(* Logix 5000 project; controller ABB_Drive_Test vendor 1 type 14 code 149 rev 33.12; software revision 33.01; part 3 of 6 *)
(* tags used below, declared in another part *)
   CF0x3MSG : MESSAGE;   // detect card
   CF0x4fMSG : MESSAGE;   // read from file
   CF0x50MSG : MESSAGE;   // write to file
   CF0x52MSG : MESSAGE;   // file open
   CF0x53MSG : MESSAGE;   // set file pointer
   CF0x54MSG : MESSAGE;   // file close
   CF0x55MSG : MESSAGE;   // delete file
   CF0x56MSG : MESSAGE;   // create directory
   CF0x57MSG : MESSAGE;   // rename/move file
   CF0x58MSG : MESSAGE;   // Find first file
   CF0x59MSG : MESSAGE;   // Find next file
   CF0x5aMSG : MESSAGE;   // Find close
   CF_data : SINT[512];
   CF_RW_functions : CF_functions;

PROGRAM CF_FunctionsProgram   (* main routine MainRoutine *)
// version 3
// june 2014
VAR
   append : BOOL := 1;
   bytestring : STRING := ' KB';
   CF_del : TIMER := (PRE := 5);
   cmd_timeout : TIMER := (PRE := 4000);
   cmdto : BOOL;
   dir_only : BOOL;
   extra_info : BOOL;
   f_nr : DINT := 75;
   falctrl01 : CONTROL := (LEN := 81, POS := 80, EN := 1, DN := 1);
   filehandle : DINT;
   flush_delay : TIMER := (PRE := 500);
   intsource : INT[100] := ([0] := 24, [1] := 76, [2] := 111, [3] := 103, [4] := 95, [5] := 49, [6] := 57, [7] := 57, [8] := 56, [9] := 95, [10] := 48, [11] := 52, [12] := 95, [13] := 48, [14] := 51, [15] := 95, [16] := 48, [17] := 50, [18] := 95, [19] := 49, [20] := 49, [21] := 46, [22] := 99, [23] := 115, [24] := 118);
   MSGtriggers : DINT;
        .0   // 0x4f
        .1   // 0x50
        .10   // 0x59
        .11   // 0x5a
        .2   // 0x51
        .3   // 0x52
        .4   // 0x53
        .5   // 0x54
        .6   // 0x55
        .7   // 0x56
        .8   // 0x57
        .9   // 0x58
   next_file_response : FS_response := (pot_holder := -242345696, fflags := 16#0000_0020, create_TS := 125357957340000000, last_write_TS := 125357957340000000, size := 252800, name[0] := '$00$18', name[1] := '$00L', name[2] := '$00o', name[3] := '$00g', name[4] := '$00_', name[5] := '$001', name[6] := '$009', name[7] := '$009', name[8] := '$008', name[9] := '$00_', name[10] := '$000', name[11] := '$003', name[12] := '$00_', name[13] := '$003', name[14] := '$001', name[15] := '$00_', name[16] := '$000', name[17] := '$004', name[18] := '$00_', name[19] := '$005', name[20] := '$005', name[21] := '$00.', name[22] := '$00c', name[23] := '$00s', name[24] := '$00v', name[25] := '$00s', name[26] := '$00v', name[27] := '8,', name[28] := '0.', name[29] := '00', name[30] := '00', name[31] := '00', name[32] := ',0', name[33] := '.9', name[34] := '00', name[35] := '00', name[36] := '00', name[37] := '00', name[38] := '1,', name[39] := '.0', name[40] := '00', name[41] := '00', name[42] := '00', name[43] := ',0', name[44] := '11', name[45] := '0.', name[46] := '00', name[47] := '00', name[48] := '00', name[49] := '1,', name[50] := '.2', name[51] := '00', name[52] := '00', name[53] := '00', name[54] := ',0',
        name[55] := '.1', name[56] := '00', name[57] := '00', name[58] := '00', name[59] := '00', name[60] := '$0A$0D', name[61] := '53', name[62] := '88', name[63] := ',8', name[64] := '.0', name[65] := '90', name[66] := '31', name[67] := '71', name[68] := '07', name[69] := '2,', name[70] := '0.', name[71] := '00', name[72] := '00', name[73] := '00', name[74] := ',0', name[75] := '.5', name[76] := '00', name[77] := '00', name[78] := '00', name[79] := '00', name[80] := '6,', name[81] := '0.', name[82] := '00', name[83] := '00', name[84] := '00', name[85] := ',0', name[86] := '.7', name[87] := '00', name[88] := '00', name[89] := '00', name[90] := '00', name[91] := '8,', name[92] := '0.', name[93] := '00', name[94] := '00', name[95] := '00', name[96] := ',0', name[97] := '.9', name[98] := '00', name[99] := '00');
        .fflags.0   // Read Only
        .fflags.1   // Hidden
        .fflags.2   // System
   prev_index : DINT := 10;
   searchstring : STRING := 'Log_1998_04_03_02_11.csv';
   slot_number : DINT;
   spacestring : STRING := '        ';
   step : DINT;
   step_copy : DINT := 99;
   tempDINT : DINT := 392;
   tempDINTAR : DINT[10] := ([0] := 1073741824, [3] := 4, [4] := 128, [7] := 40, [8] := 20224);
   tempstring : STRING := '$01$00';
END_VAR

ROUTINE ascii2uni   (* ladder *)
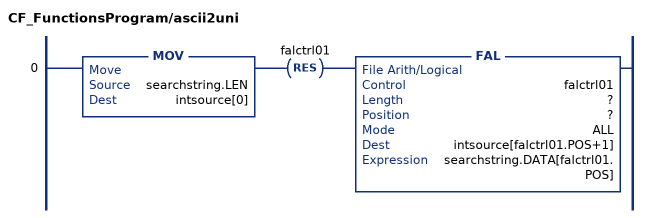
   0: MOV(searchstring.LEN,intsource[0])RES(falctrl01)FAL(falctrl01,?,?,ALL,intsource[falctrl01.POS+1],searchstring.DATA[falctrl01.POS]);
END_ROUTINE

ROUTINE MainRoutine   (* ladder *)
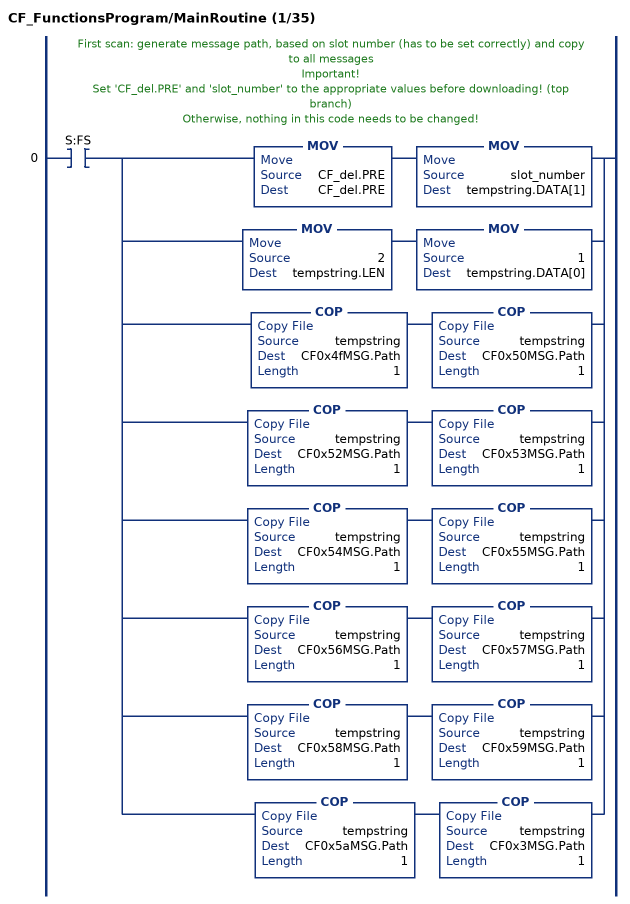
   // First scan: generate message path, based on slot number (has to be set correctly) and copy to all messages
   // Important!
   // Set 'CF_del.PRE' and 'slot_number' to the appropriate values before downloading! (top branch)
   // Otherwise, nothing in this code needs to be changed!
   0: XIC(S:FS)[MOV(CF_del.PRE,CF_del.PRE) MOV(slot_number,tempstring.DATA[1]) ,MOV(2,tempstring.LEN) MOV(1,tempstring.DATA[0]) ,COP(tempstring,CF0x4fMSG.Path,1) COP(tempstring,CF0x50MSG.Path,1) ,COP(tempstring,CF0x52MSG.Path,1) COP(tempstring,CF0x53MSG.Path,1) ,COP(tempstring,CF0x54MSG.Path,1) COP(tempstring,CF0x55MSG.Path,1) ,COP(tempstring,CF0x56MSG.Path,1) COP(tempstring,CF0x57MSG.Path,1) ,COP(tempstring,CF0x58MSG.Path,1) COP(tempstring,CF0x59MSG.Path,1) ,COP(tempstring,CF0x5aMSG.Path,1) COP(tempstring,CF0x3MSG.Path,1) ];
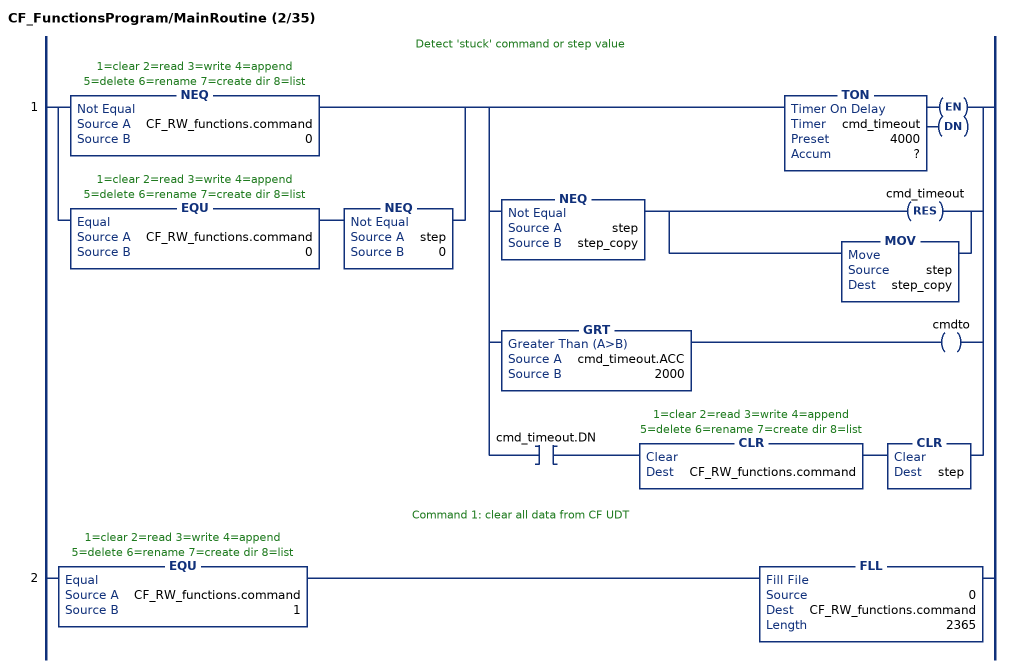
   // Detect 'stuck' command or step value
   1: [NEQ(CF_RW_functions.command,0) ,EQU(CF_RW_functions.command,0) NEQ(step,0) ][TON(cmd_timeout,?,?) ,NEQ(step,step_copy) [RES(cmd_timeout) ,MOV(step,step_copy) ] ,GRT(cmd_timeout.ACC,2000) OTE(cmdto) ,XIC(cmd_timeout.DN) CLR(CF_RW_functions.command) CLR(step) ];
   // Command 1: clear all data from CF UDT
   2: EQU(CF_RW_functions.command,1)FLL(0,CF_RW_functions.command,2365);
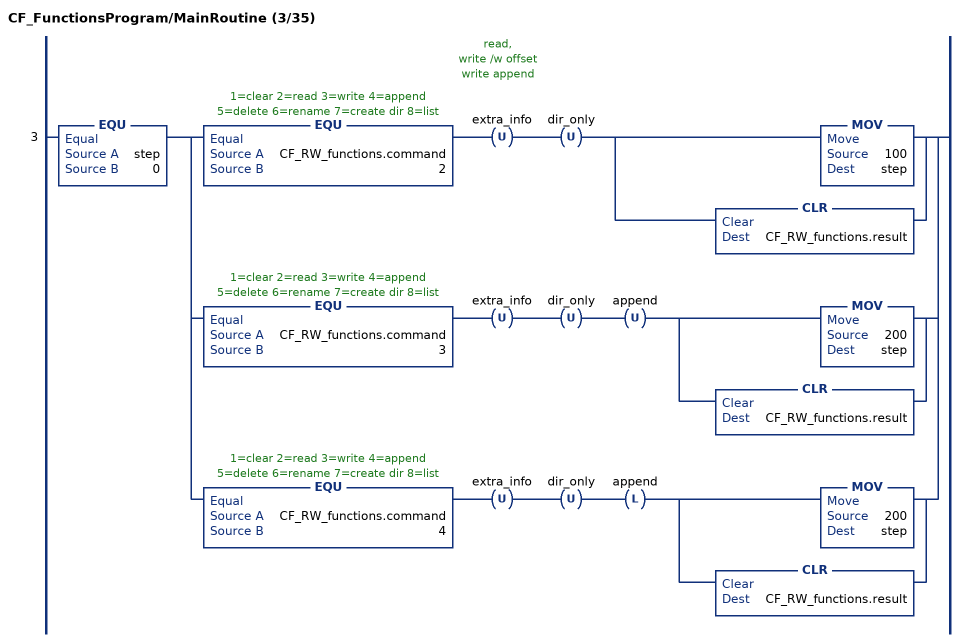
   // read,
   // write /w offset
   // write append
   3: EQU(step,0)[EQU(CF_RW_functions.command,2) OTU(extra_info) OTU(dir_only) [MOV(100,step) ,CLR(CF_RW_functions.result) ] ,EQU(CF_RW_functions.command,3) OTU(extra_info) OTU(dir_only) OTU(append) [MOV(200,step) ,CLR(CF_RW_functions.result) ] ,EQU(CF_RW_functions.command,4) OTU(extra_info) OTU(dir_only) OTL(append) [MOV(200,step) ,CLR(CF_RW_functions.result) ] ];
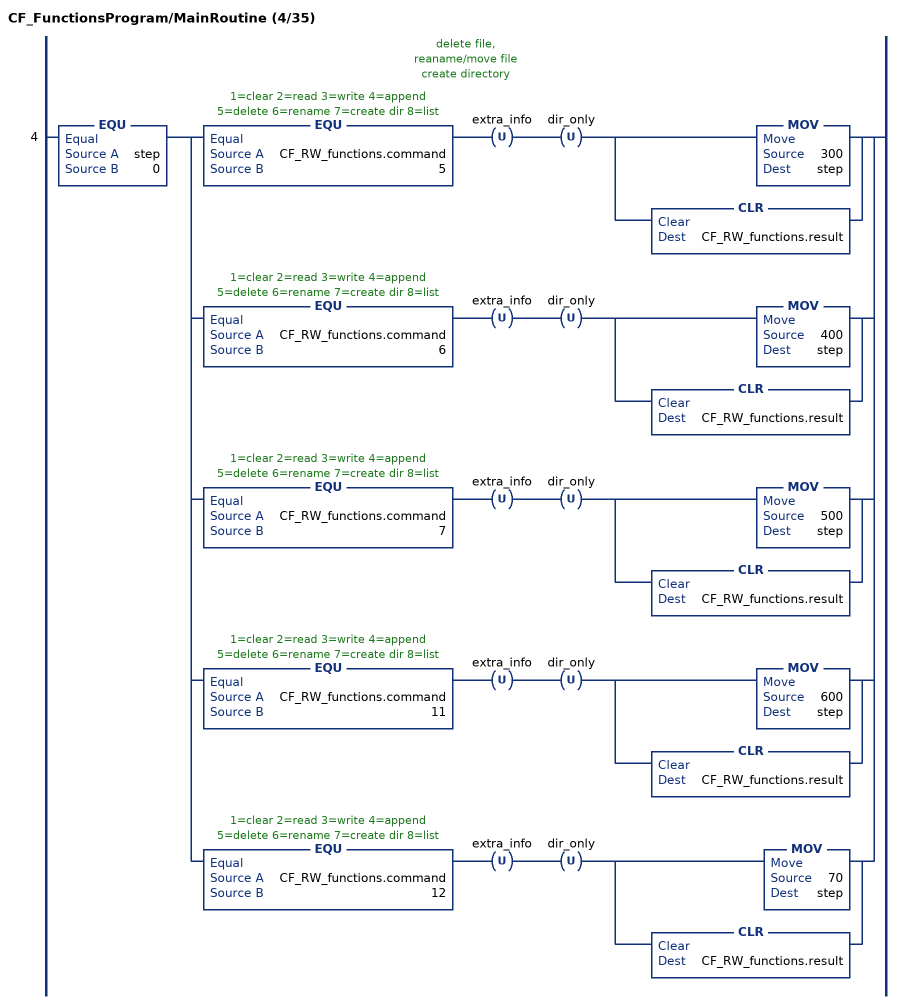
   // delete file,
   // reaname/move file
   // create directory
   4: EQU(step,0)[EQU(CF_RW_functions.command,5) OTU(extra_info) OTU(dir_only) [MOV(300,step) ,CLR(CF_RW_functions.result) ] ,EQU(CF_RW_functions.command,6) OTU(extra_info) OTU(dir_only) [MOV(400,step) ,CLR(CF_RW_functions.result) ] ,EQU(CF_RW_functions.command,7) OTU(extra_info) OTU(dir_only) [MOV(500,step) ,CLR(CF_RW_functions.result) ] ,EQU(CF_RW_functions.command,11) OTU(extra_info) OTU(dir_only) [MOV(600,step) ,CLR(CF_RW_functions.result) ] ,EQU(CF_RW_functions.command,12) OTU(extra_info) OTU(dir_only) [MOV(70,step) ,CLR(CF_RW_functions.result) ] ];
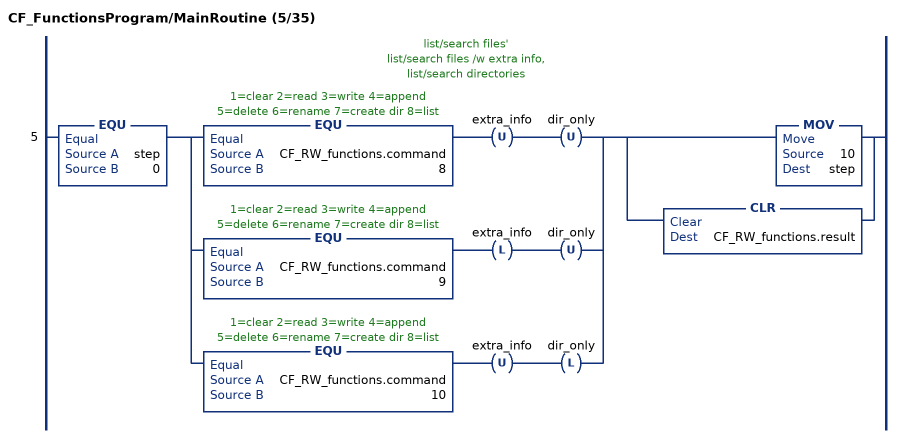
   // list/search files'
   // list/search files /w extra info,
   // list/search directories
   5: EQU(step,0)[EQU(CF_RW_functions.command,8) OTU(extra_info) OTU(dir_only) ,EQU(CF_RW_functions.command,9) OTL(extra_info) OTU(dir_only) ,EQU(CF_RW_functions.command,10) OTU(extra_info) OTL(dir_only) ][MOV(10,step) ,CLR(CF_RW_functions.result) ];
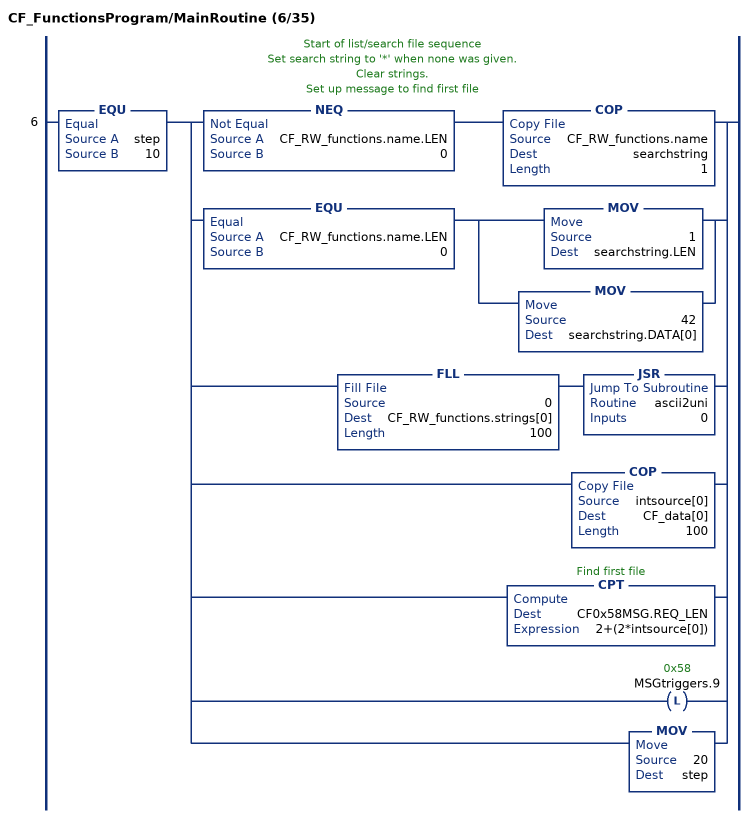
   // Start of list/search file sequence
   //  Set search string to '*' when none was given.
   // Clear strings.
   // Set up message to find first file
   6: EQU(step,10)[NEQ(CF_RW_functions.name.LEN,0) COP(CF_RW_functions.name,searchstring,1) ,EQU(CF_RW_functions.name.LEN,0) [MOV(1,searchstring.LEN) ,MOV(42,searchstring.DATA[0]) ] ,FLL(0,CF_RW_functions.strings[0],100) JSR(ascii2uni,0) ,COP(intsource[0],CF_data[0],100) ,CPT(CF0x58MSG.REQ_LEN,2+(2*intsource[0])) ,OTL(MSGtriggers.9) ,MOV(20,step) ];
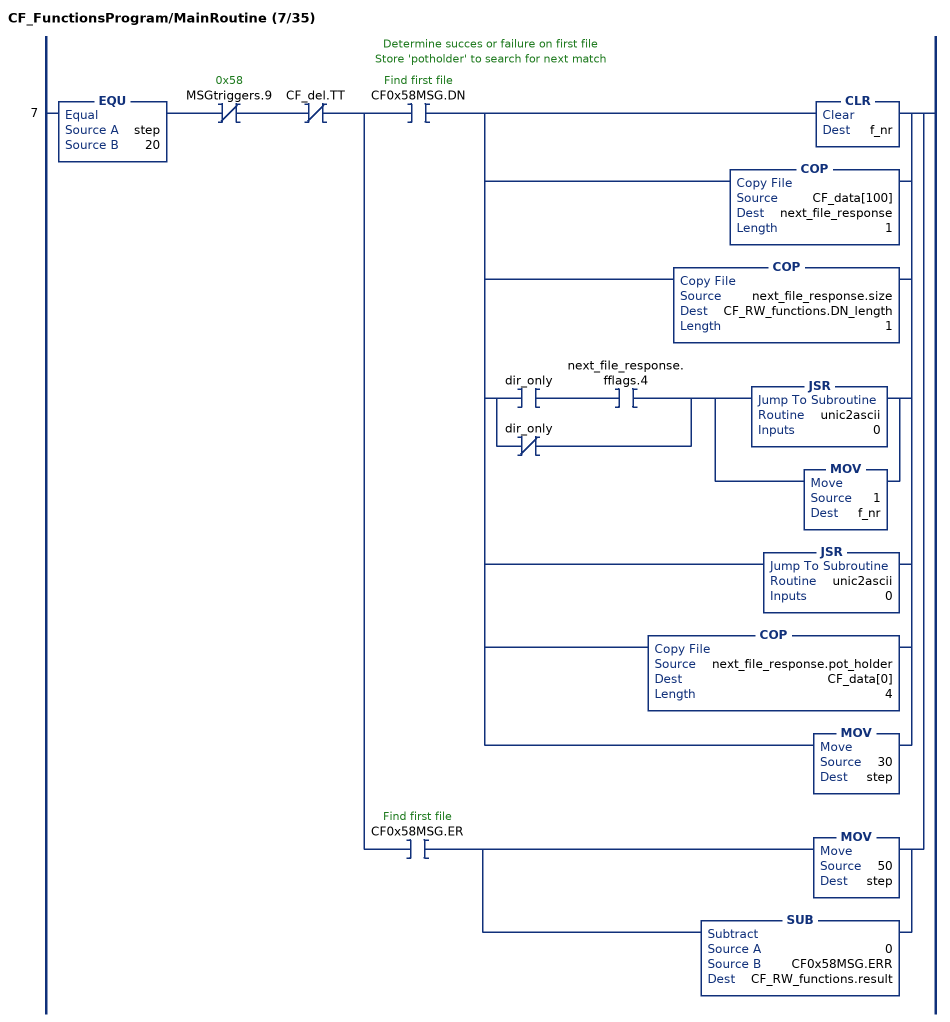
   // Determine succes or failure on first file
   // Store 'potholder' to search for next match
   7: EQU(step,20)XIO(MSGtriggers.9)XIO(CF_del.TT)[XIC(CF0x58MSG.DN) [CLR(f_nr) ,COP(CF_data[100],next_file_response,1) ,COP(next_file_response.size,CF_RW_functions.DN_length,1) ,[XIC(dir_only) XIC(next_file_response.fflags.4) ,XIO(dir_only) ] [JSR(unic2ascii,0) ,MOV(1,f_nr) ] ,JSR(unic2ascii,0) ,COP(next_file_response.pot_holder,CF_data[0],4) ,MOV(30,step) ] ,XIC(CF0x58MSG.ER) [MOV(50,step) ,SUB(0,CF0x58MSG.ERR,CF_RW_functions.result) ] ];
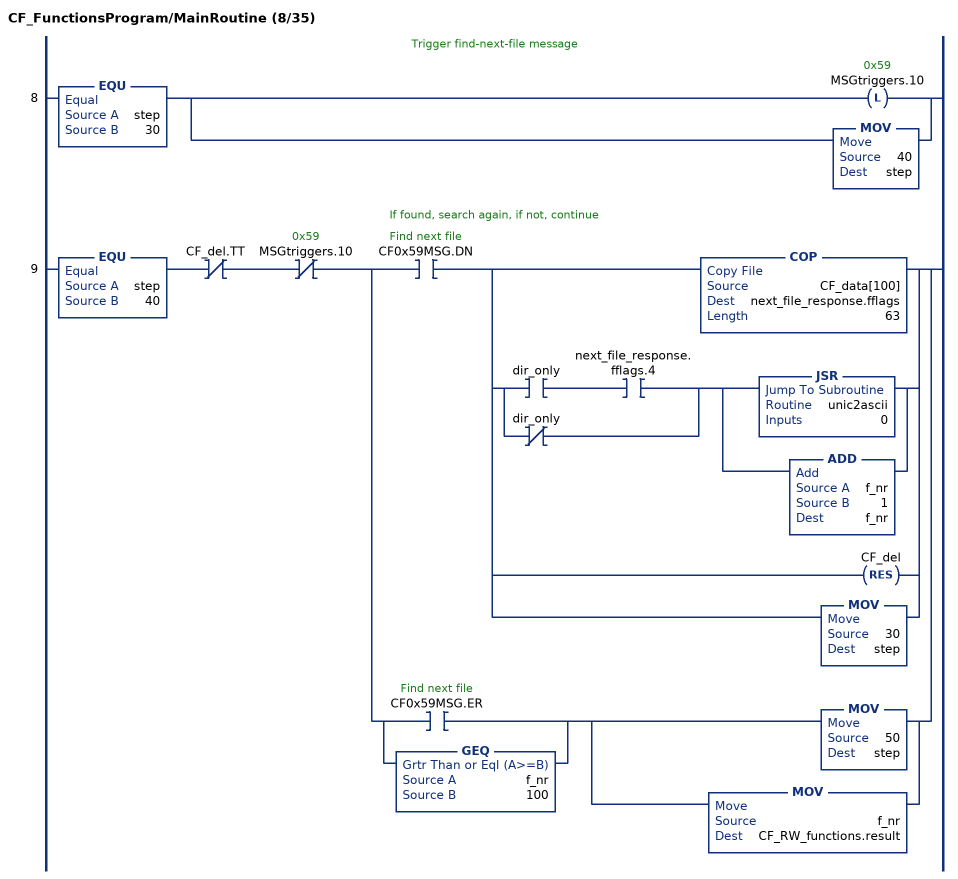
   // Trigger find-next-file message
   8: EQU(step,30)[OTL(MSGtriggers.10) ,MOV(40,step) ];
   // If found, search again, if not, continue
   9: EQU(step,40)XIO(CF_del.TT)XIO(MSGtriggers.10)[XIC(CF0x59MSG.DN) [COP(CF_data[100],next_file_response.fflags,63) ,[XIC(dir_only) XIC(next_file_response.fflags.4) ,XIO(dir_only) ] [JSR(unic2ascii,0) ,ADD(f_nr,1,f_nr) ] ,RES(CF_del) ,MOV(30,step) ] ,[XIC(CF0x59MSG.ER) ,GEQ(f_nr,100) ] [MOV(50,step) ,MOV(f_nr,CF_RW_functions.result) ] ];
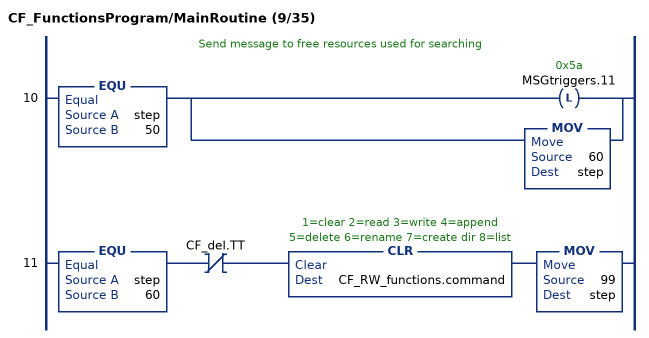
   // Send message to free resources used for searching
   10: EQU(step,50)[OTL(MSGtriggers.11) ,MOV(60,step) ];
   11: EQU(step,60)XIO(CF_del.TT)CLR(CF_RW_functions.command)MOV(99,step);
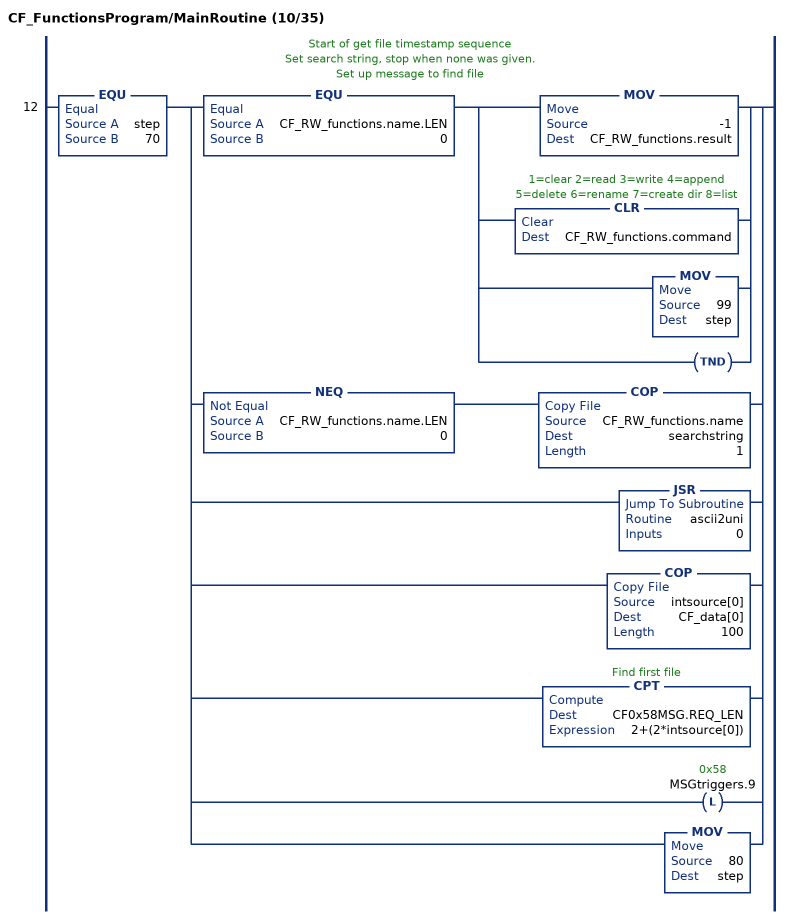
   // Start of get file timestamp sequence
   //  Set search string, stop when none was given.
   // Set up message to find file
   12: EQU(step,70)[EQU(CF_RW_functions.name.LEN,0) [MOV(-1,CF_RW_functions.result) ,CLR(CF_RW_functions.command) ,MOV(99,step) ,TND() ] ,NEQ(CF_RW_functions.name.LEN,0) COP(CF_RW_functions.name,searchstring,1) ,JSR(ascii2uni,0) ,COP(intsource[0],CF_data[0],100) ,CPT(CF0x58MSG.REQ_LEN,2+(2*intsource[0])) ,OTL(MSGtriggers.9) ,MOV(80,step) ];
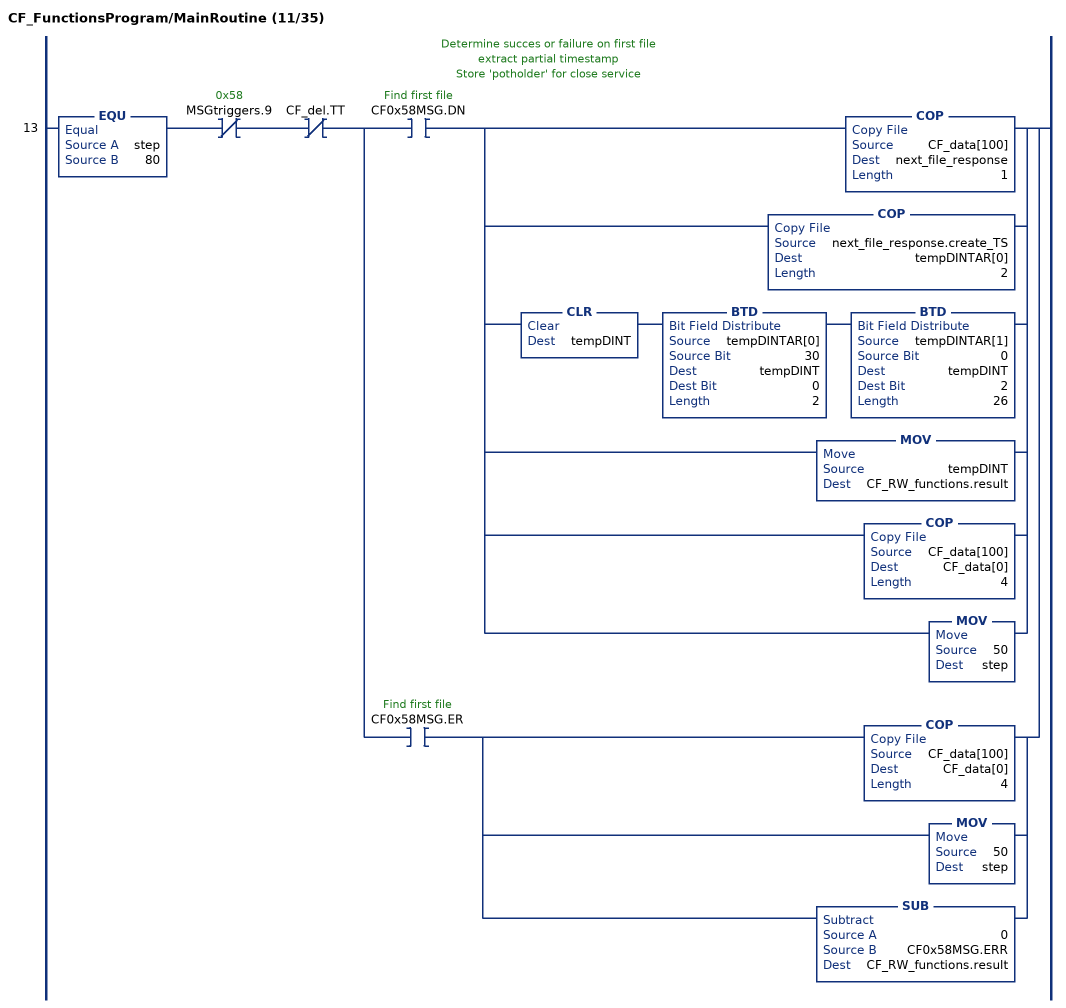
   // Determine succes or failure on first file
   // extract partial timestamp
   // Store 'potholder' for close service
   13: EQU(step,80)XIO(MSGtriggers.9)XIO(CF_del.TT)[XIC(CF0x58MSG.DN) [COP(CF_data[100],next_file_response,1) ,COP(next_file_response.create_TS,tempDINTAR[0],2) ,CLR(tempDINT) BTD(tempDINTAR[0],30,tempDINT,0,2) BTD(tempDINTAR[1],0,tempDINT,2,26) ,MOV(tempDINT,CF_RW_functions.result) ,COP(CF_data[100],CF_data[0],4) ,MOV(50,step) ] ,XIC(CF0x58MSG.ER) [COP(CF_data[100],CF_data[0],4) ,MOV(50,step) ,SUB(0,CF0x58MSG.ERR,CF_RW_functions.result) ] ];
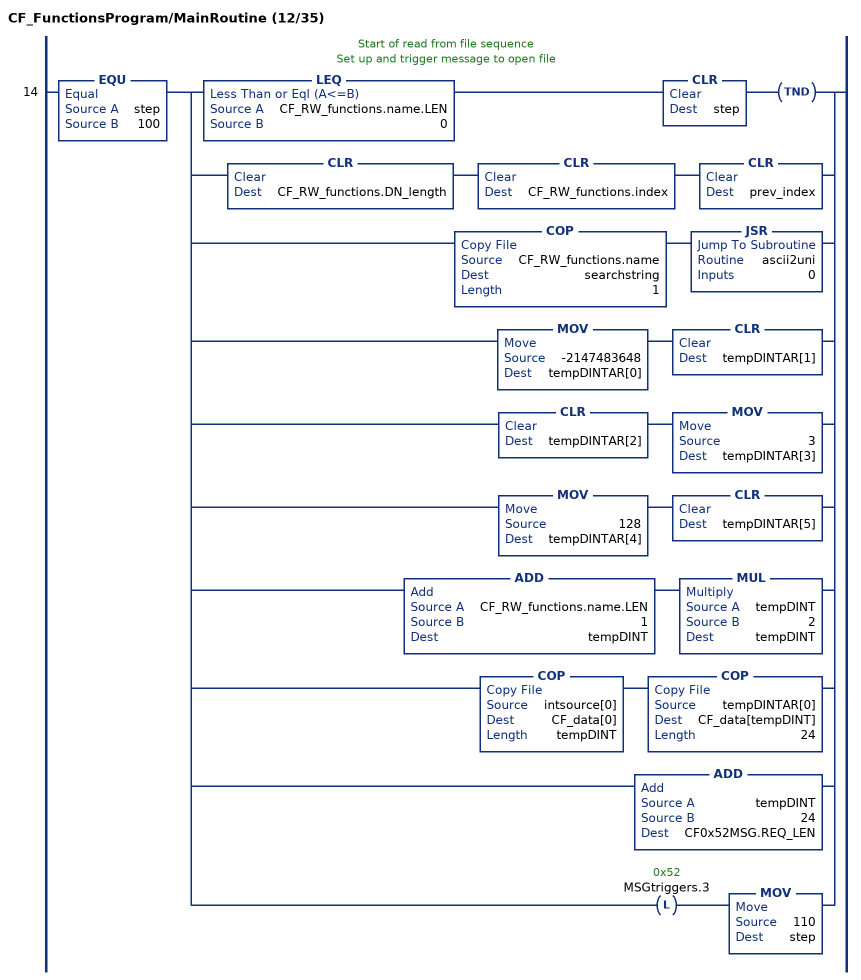
   // Start of read from file sequence
   // Set up and trigger message to open file
   14: EQU(step,100)[LEQ(CF_RW_functions.name.LEN,0) CLR(step) TND() ,CLR(CF_RW_functions.DN_length) CLR(CF_RW_functions.index) CLR(prev_index) ,COP(CF_RW_functions.name,searchstring,1) JSR(ascii2uni,0) ,MOV(-2147483648,tempDINTAR[0]) CLR(tempDINTAR[1]) ,CLR(tempDINTAR[2]) MOV(3,tempDINTAR[3]) ,MOV(128,tempDINTAR[4]) CLR(tempDINTAR[5]) ,ADD(CF_RW_functions.name.LEN,1,tempDINT) MUL(tempDINT,2,tempDINT) ,COP(intsource[0],CF_data[0],tempDINT) COP(tempDINTAR[0],CF_data[tempDINT],24) ,ADD(tempDINT,24,CF0x52MSG.REQ_LEN) ,OTL(MSGtriggers.3) MOV(110,step) ];
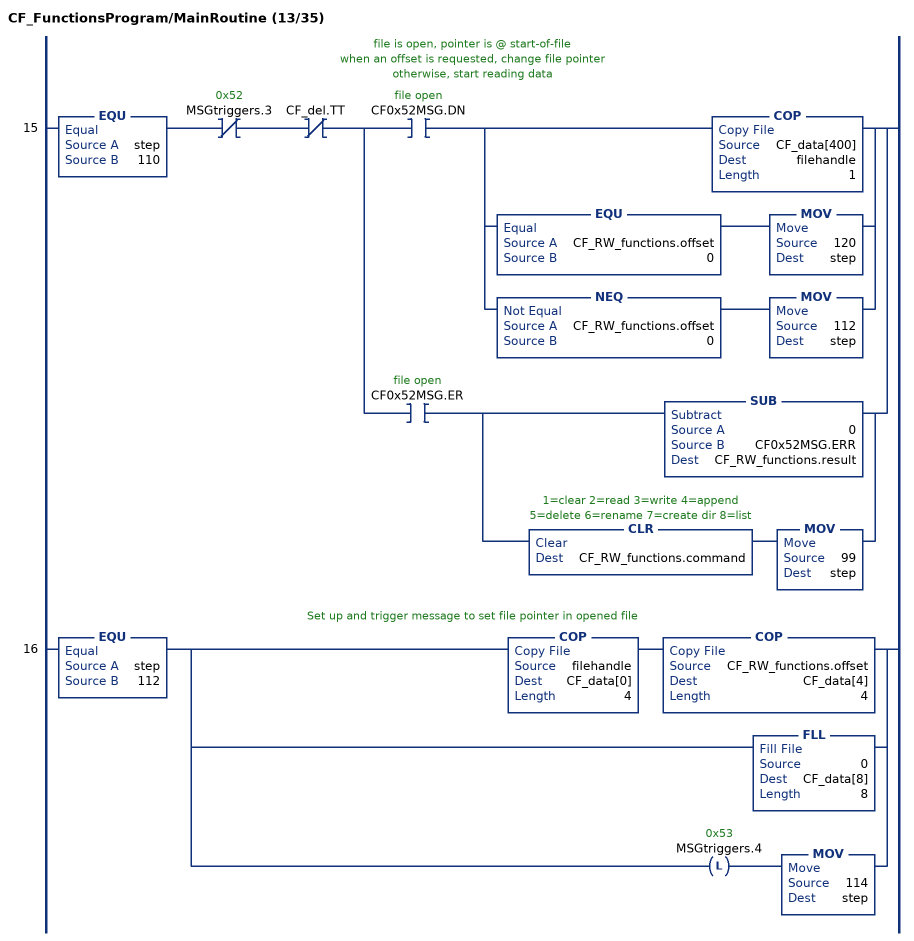
   // file is open, pointer is @ start-of-file
   // when an offset is requested, change file pointer
   // otherwise, start reading data
   15: EQU(step,110)XIO(MSGtriggers.3)XIO(CF_del.TT)[XIC(CF0x52MSG.DN) [COP(CF_data[400],filehandle,1) ,EQU(CF_RW_functions.offset,0) MOV(120,step) ,NEQ(CF_RW_functions.offset,0) MOV(112,step) ] ,XIC(CF0x52MSG.ER) [SUB(0,CF0x52MSG.ERR,CF_RW_functions.result) ,CLR(CF_RW_functions.command) MOV(99,step) ] ];
   // Set up and trigger message to set file pointer in opened file
   16: EQU(step,112)[COP(filehandle,CF_data[0],4) COP(CF_RW_functions.offset,CF_data[4],4) ,FLL(0,CF_data[8],8) ,OTL(MSGtriggers.4) MOV(114,step) ];
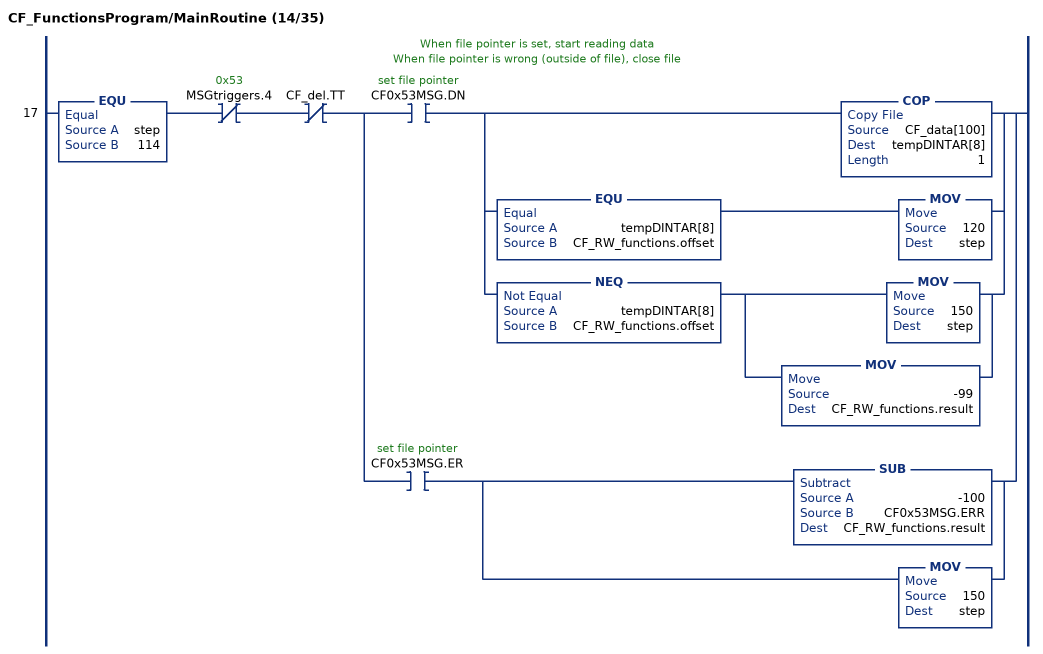
   // When file pointer is set, start reading data
   // When file pointer is wrong (outside of file), close file
   17: EQU(step,114)XIO(MSGtriggers.4)XIO(CF_del.TT)[XIC(CF0x53MSG.DN) [COP(CF_data[100],tempDINTAR[8],1) ,EQU(tempDINTAR[8],CF_RW_functions.offset) MOV(120,step) ,NEQ(tempDINTAR[8],CF_RW_functions.offset) [MOV(150,step) ,MOV(-99,CF_RW_functions.result) ] ] ,XIC(CF0x53MSG.ER) [SUB(-100,CF0x53MSG.ERR,CF_RW_functions.result) ,MOV(150,step) ] ];
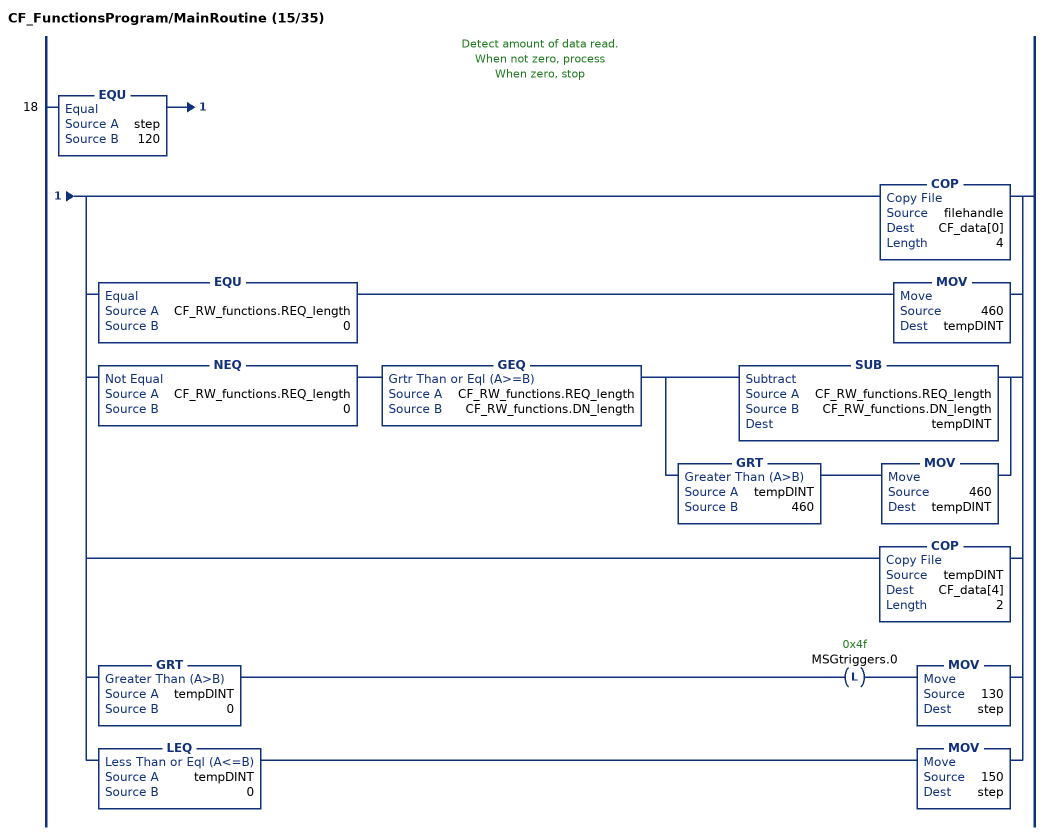
   // Detect amount of data read.
   // When not zero, process
   // When zero, stop
   18: EQU(step,120)[COP(filehandle,CF_data[0],4) ,EQU(CF_RW_functions.REQ_length,0) MOV(460,tempDINT) ,NEQ(CF_RW_functions.REQ_length,0) GEQ(CF_RW_functions.REQ_length,CF_RW_functions.DN_length) [SUB(CF_RW_functions.REQ_length,CF_RW_functions.DN_length,tempDINT) ,GRT(tempDINT,460) MOV(460,tempDINT) ] ,COP(tempDINT,CF_data[4],2) ,GRT(tempDINT,0) OTL(MSGtriggers.0) MOV(130,step) ,LEQ(tempDINT,0) MOV(150,step) ];
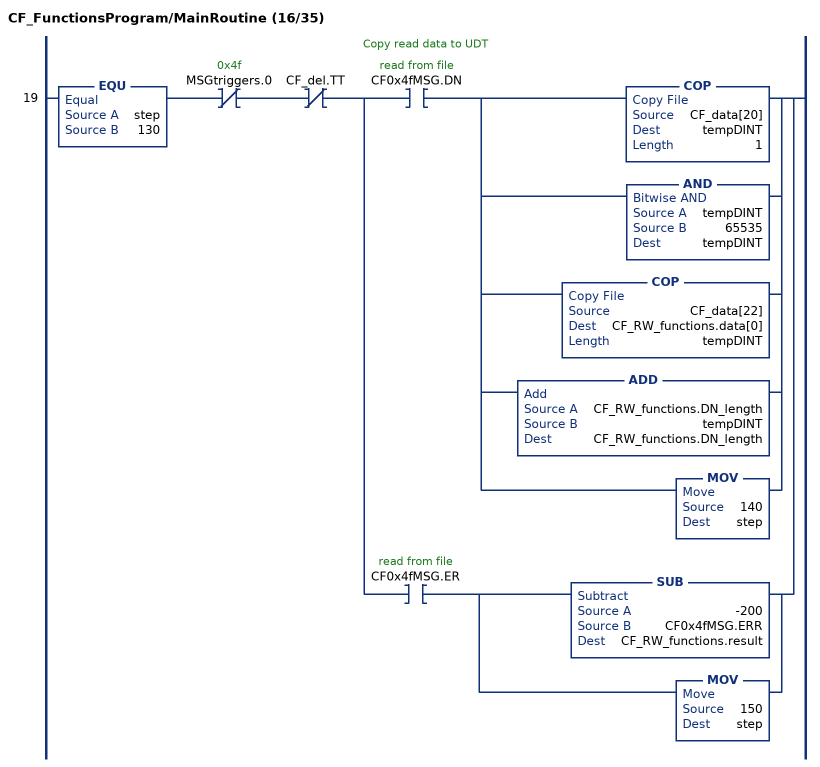
   // Copy read data to UDT
   19: EQU(step,130)XIO(MSGtriggers.0)XIO(CF_del.TT)[XIC(CF0x4fMSG.DN) [COP(CF_data[20],tempDINT,1) ,AND(tempDINT,65535,tempDINT) ,COP(CF_data[22],CF_RW_functions.data[0],tempDINT) ,ADD(CF_RW_functions.DN_length,tempDINT,CF_RW_functions.DN_length) ,MOV(140,step) ] ,XIC(CF0x4fMSG.ER) [SUB(-200,CF0x4fMSG.ERR,CF_RW_functions.result) ,MOV(150,step) ] ];
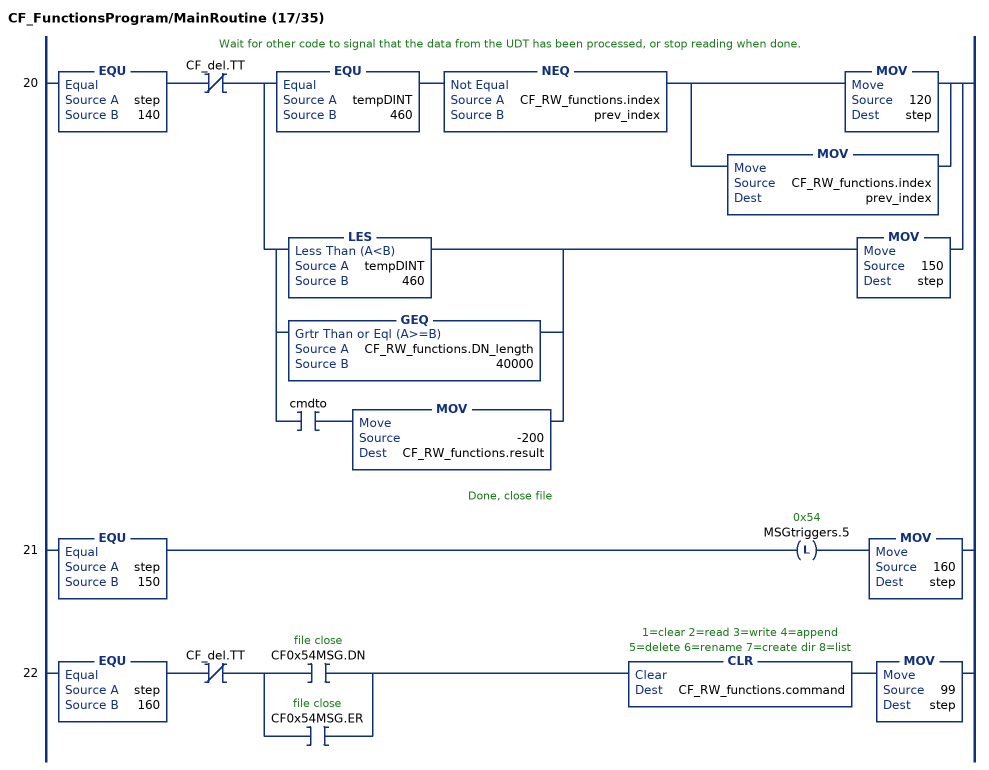
   // Wait for other code to signal that the data from the UDT has been processed, or stop reading when done.
   20: EQU(step,140)XIO(CF_del.TT)[EQU(tempDINT,460) NEQ(CF_RW_functions.index,prev_index) [MOV(120,step) ,MOV(CF_RW_functions.index,prev_index) ] ,[LES(tempDINT,460) ,GEQ(CF_RW_functions.DN_length,40000) ,XIC(cmdto) MOV(-200,CF_RW_functions.result) ] MOV(150,step) ];
   // Done, close file
   21: EQU(step,150)OTL(MSGtriggers.5)MOV(160,step);
   22: EQU(step,160)XIO(CF_del.TT)[XIC(CF0x54MSG.DN) ,XIC(CF0x54MSG.ER) ]CLR(CF_RW_functions.command)MOV(99,step);
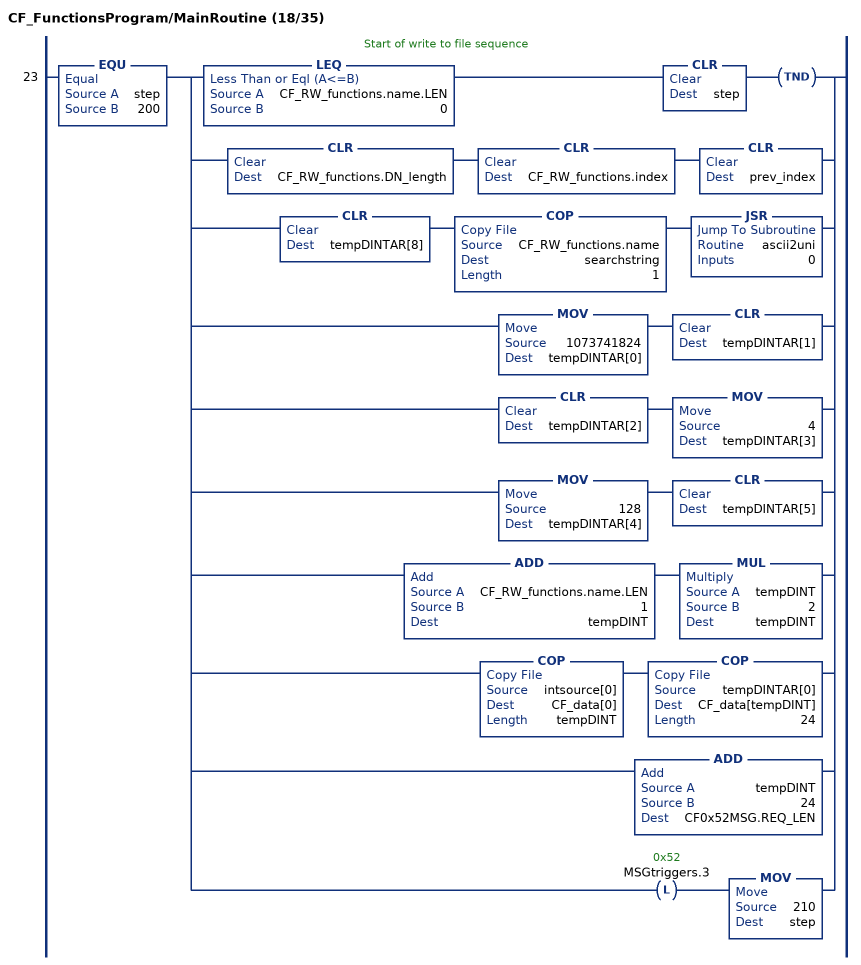
   // Start of write to file sequence
   23: EQU(step,200)[LEQ(CF_RW_functions.name.LEN,0) CLR(step) TND() ,CLR(CF_RW_functions.DN_length) CLR(CF_RW_functions.index) CLR(prev_index) ,CLR(tempDINTAR[8]) COP(CF_RW_functions.name,searchstring,1) JSR(ascii2uni,0) ,MOV(1073741824,tempDINTAR[0]) CLR(tempDINTAR[1]) ,CLR(tempDINTAR[2]) MOV(4,tempDINTAR[3]) ,MOV(128,tempDINTAR[4]) CLR(tempDINTAR[5]) ,ADD(CF_RW_functions.name.LEN,1,tempDINT) MUL(tempDINT,2,tempDINT) ,COP(intsource[0],CF_data[0],tempDINT) COP(tempDINTAR[0],CF_data[tempDINT],24) ,ADD(tempDINT,24,CF0x52MSG.REQ_LEN) ,OTL(MSGtriggers.3) MOV(210,step) ];
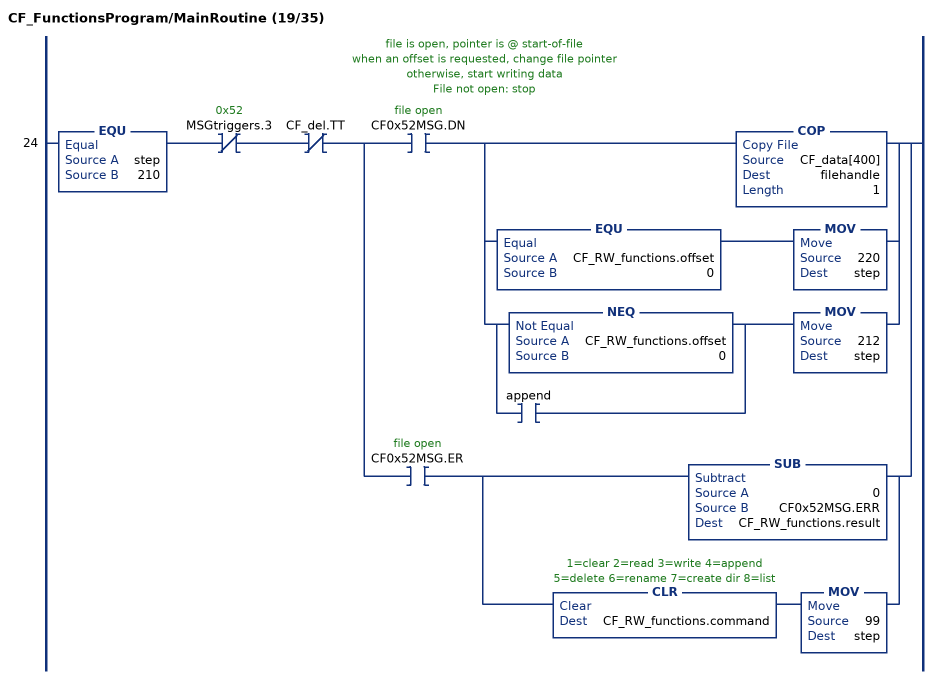
   // file is open, pointer is @ start-of-file
   // when an offset is requested, change file pointer
   // otherwise, start writing data
   // File not open: stop
   24: EQU(step,210)XIO(MSGtriggers.3)XIO(CF_del.TT)[XIC(CF0x52MSG.DN) [COP(CF_data[400],filehandle,1) ,EQU(CF_RW_functions.offset,0) MOV(220,step) ,[NEQ(CF_RW_functions.offset,0) ,XIC(append) ] MOV(212,step) ] ,XIC(CF0x52MSG.ER) [SUB(0,CF0x52MSG.ERR,CF_RW_functions.result) ,CLR(CF_RW_functions.command) MOV(99,step) ] ];
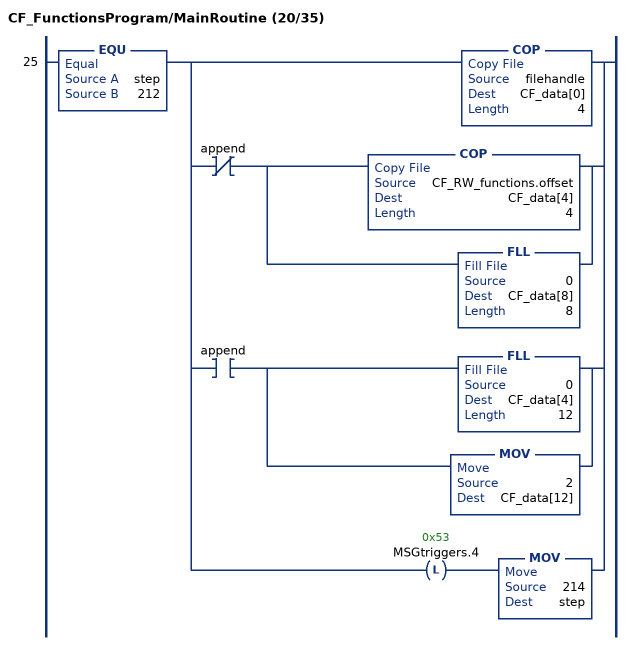
   25: EQU(step,212)[COP(filehandle,CF_data[0],4) ,XIO(append) [COP(CF_RW_functions.offset,CF_data[4],4) ,FLL(0,CF_data[8],8) ] ,XIC(append) [FLL(0,CF_data[4],12) ,MOV(2,CF_data[12]) ] ,OTL(MSGtriggers.4) MOV(214,step) ];
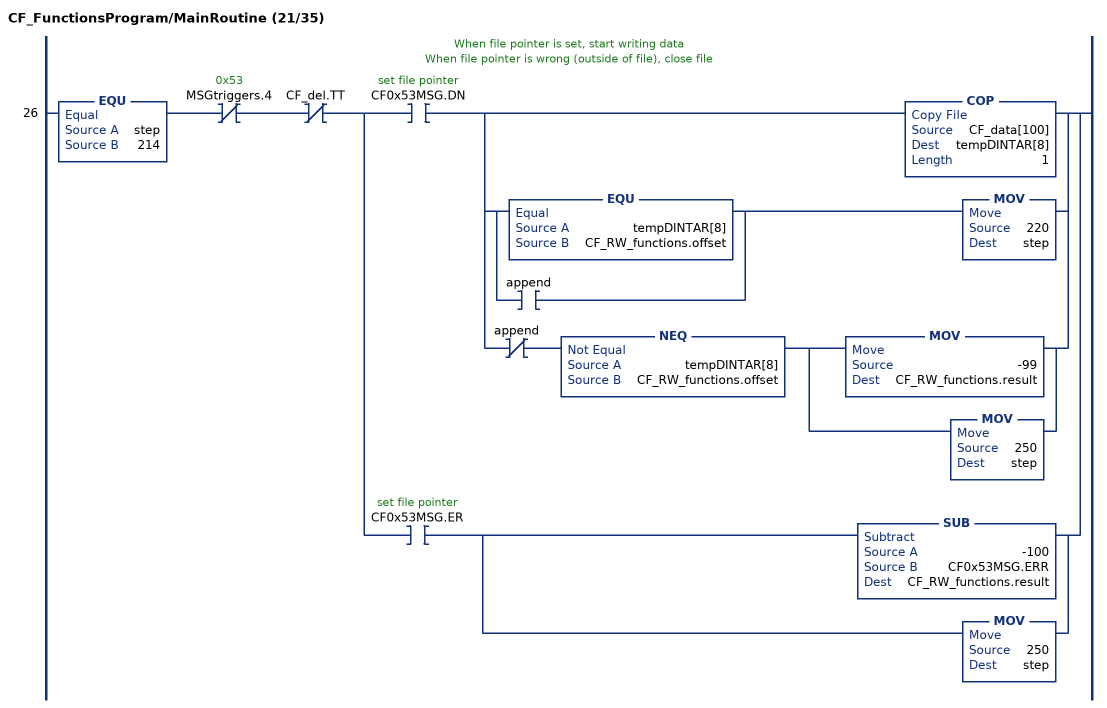
   // When file pointer is set, start writing data
   // When file pointer is wrong (outside of file), close file
   26: EQU(step,214)XIO(MSGtriggers.4)XIO(CF_del.TT)[XIC(CF0x53MSG.DN) [COP(CF_data[100],tempDINTAR[8],1) ,[EQU(tempDINTAR[8],CF_RW_functions.offset) ,XIC(append) ] MOV(220,step) ,XIO(append) NEQ(tempDINTAR[8],CF_RW_functions.offset) [MOV(-99,CF_RW_functions.result) ,MOV(250,step) ] ] ,XIC(CF0x53MSG.ER) [SUB(-100,CF0x53MSG.ERR,CF_RW_functions.result) ,MOV(250,step) ] ];
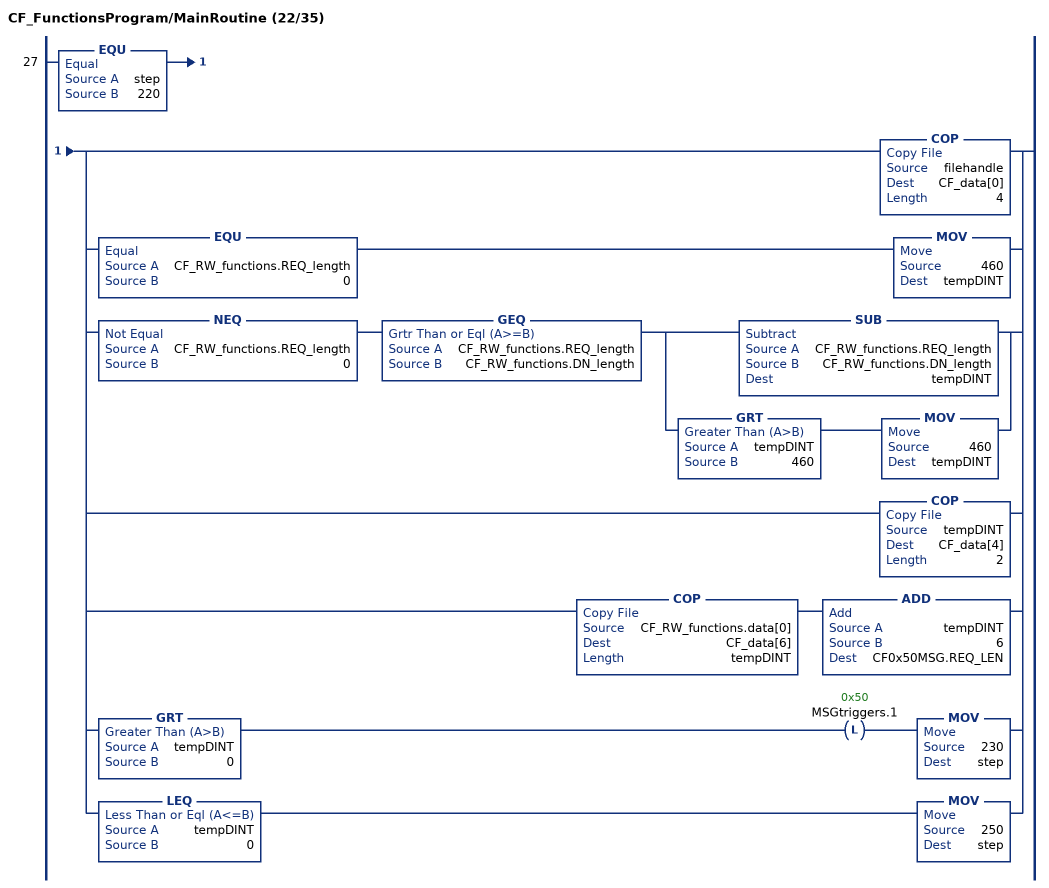
   27: EQU(step,220)[COP(filehandle,CF_data[0],4) ,EQU(CF_RW_functions.REQ_length,0) MOV(460,tempDINT) ,NEQ(CF_RW_functions.REQ_length,0) GEQ(CF_RW_functions.REQ_length,CF_RW_functions.DN_length) [SUB(CF_RW_functions.REQ_length,CF_RW_functions.DN_length,tempDINT) ,GRT(tempDINT,460) MOV(460,tempDINT) ] ,COP(tempDINT,CF_data[4],2) ,COP(CF_RW_functions.data[0],CF_data[6],tempDINT) ADD(tempDINT,6,CF0x50MSG.REQ_LEN) ,GRT(tempDINT,0) OTL(MSGtriggers.1) MOV(230,step) ,LEQ(tempDINT,0) MOV(250,step) ];
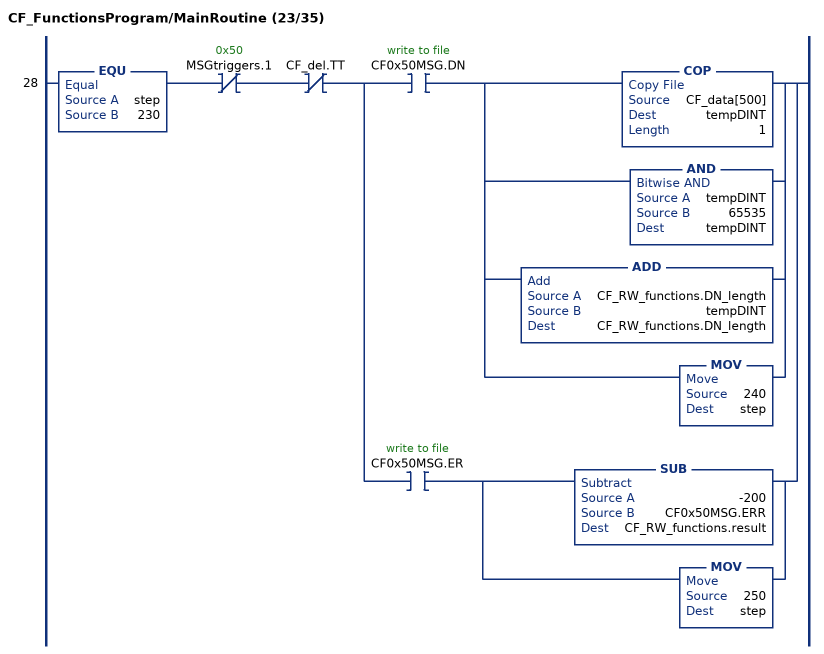
   28: EQU(step,230)XIO(MSGtriggers.1)XIO(CF_del.TT)[XIC(CF0x50MSG.DN) [COP(CF_data[500],tempDINT,1) ,AND(tempDINT,65535,tempDINT) ,ADD(CF_RW_functions.DN_length,tempDINT,CF_RW_functions.DN_length) ,MOV(240,step) ] ,XIC(CF0x50MSG.ER) [SUB(-200,CF0x50MSG.ERR,CF_RW_functions.result) ,MOV(250,step) ] ];
